// TIA Portal V20 export
// export: Created 2025-12-01T14:57:26.5426352Z, ExportSetting None, DisplayName Totally Integrated Automation Portal, DisplayVersion V20 Update 3, DisplayName TIA Portal Openness, DisplayVersion V20 Update 3, DisplayName TIA Portal Version Control Interface, DisplayVersion V20 Update 3, DisplayName STEP 7 Professional, DisplayVersion V20 Update 3, DisplayName STEP 7 Safety, DisplayVersion V20 Update 2, DisplayName WinCC Basic/Comfort/Advanced, DisplayVersion V20 Update 3, DisplayName WinCC Professional, DisplayVersion V20 Update 3, DisplayName WinCC Unified, DisplayVersion V20 Update 3
FUNCTION "FC600_ini+ref_dato_encoder_NEW" : Void   // FC600, LAD
{ S7_Optimized_Access := 'FALSE' }
// stored: AutoNumber false, SetENOAutomatically false
   VAR_INPUT
      Detector_referencia : Bool;
      ID_Quimarox : UInt;
      dato_encoder_actual : DInt;
      V_cnt_tout_refresco : UDInt;
   END_VAR
   VAR_IN_OUT
      m_aux_pf_detect : Bool;
      MEM_CNT_TOUT : UDInt;
   END_VAR
   VAR_TEMP
      fp_detector : Bool;
      tout : Bool;
      fecha : Date_And_Time;
      retval : Int;
      hora : Time_Of_Day;
   END_VAR
   VAR_TEMP   // added for the SCL form of the ladder/FBD networks
      _w1 : Bool;
   END_VAR
BEGIN

REGION Network 1
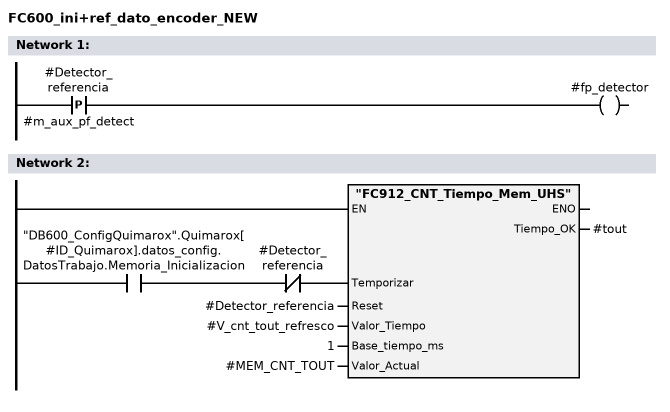
   RUNG wire#powerrail
      P_Contact(operand := #Detector_referencia, bit := #m_aux_pf_detect)
      Coil( #fp_detector )
   END_RUNG
   // the same network as SCL:
   #_w1 := #Detector_referencia AND NOT #m_aux_pf_detect;   // rising edge of #Detector_referencia
   #m_aux_pf_detect := #Detector_referencia;
   #fp_detector := #_w1;
END_REGION

REGION Network 2
   RUNG wire#powerrail
      "FC912_CNT_Tiempo_Mem_UHS"(Temporizar := wire#w1, Reset := #Detector_referencia, Valor_Tiempo := #V_cnt_tout_refresco, Base_tiempo_ms := 1, Valor_Actual := #MEM_CNT_TOUT, Tiempo_OK => #tout)
   END_RUNG
   RUNG wire#powerrail
      Contact( "DB600_ConfigQuimarox".Quimarox[#ID_Quimarox].datos_config.DatosTrabajo.Memoria_Inicializacion )
      I_Contact( #Detector_referencia )
   END_RUNG wire#w1
   // the same network as SCL:
   "FC912_CNT_Tiempo_Mem_UHS"(Temporizar := "DB600_ConfigQuimarox".Quimarox[#ID_Quimarox].datos_config.DatosTrabajo.Memoria_Inicializacion AND NOT #Detector_referencia,
                           Reset := #Detector_referencia,
                           Valor_Tiempo := #V_cnt_tout_refresco,
                           Base_tiempo_ms := 1,
                           Valor_Actual := #MEM_CNT_TOUT,
                           Tiempo_OK => #tout);
END_REGION

NETWORK
TITLE = 

      SET;
      A     "DB600_ConfigQuimarox".Quimarox[#ID_Quimarox].datos_config.DatosTrabajo.Memoria_Inicializacion;
      JC    NXT;

      SET;
      AN    #fp_detector;
      JC    fin;


NETWORK
TITLE = 
//====================================================================================================================================================================================
// primera actualización del dato del encoder. Ademas de memorizar cual es el dato del encoder en este momento y pasarlo a la memoria, registramos la hora en al que se ha producido

      L     #dato_encoder_actual;  //en el primer ciclo giramos en vacio hasta que detectemos el elemento para referenciar
      T     "DB600_ConfigQuimarox".Quimarox[#ID_Quimarox].datos_config.DatosTrabajo.Memoria_Dato_Encoder;

      SET;
      =     "DB600_ConfigQuimarox".Quimarox[#ID_Quimarox].datos_config.DatosTrabajo.Memoria_Inicializacion;

      CALL  RD_SYS_T
      ( RET_VAL := #retval,
        OUT     := #fecha
      );

      CALL  T_CONV
      ( IN  := #fecha,
        OUT := #hora
      );


      L     #hora;
      T     "DB600_ConfigQuimarox".Quimarox[#ID_Quimarox].datos_config.DatosTrabajo.Hora_Ultimo_Refresco;  //#Hora_ultimo_refresco

      BE;

//===============================================================================================================================================================================

NETWORK
TITLE = 
NXT:  A     #fp_detector;
      JC    REF;

      BE;


NETWORK
TITLE = 
//==================================================================================================================================00
REF:  L     #dato_encoder_actual;
      T     "DB600_ConfigQuimarox".Quimarox[#ID_Quimarox].datos_config.DatosTrabajo.Memoria_Dato_Encoder;

      CALL  RD_SYS_T
      ( RET_VAL := #retval,
        OUT     := #fecha
      );

      CALL  T_CONV
      ( IN  := #fecha,
        OUT := #hora
      );

      L     "DB600_ConfigQuimarox".Quimarox[#ID_Quimarox].datos_config.DatosTrabajo.Hora_Ultimo_Refresco;  //#Hora_ultimo_refresco
      T     "DB600_ConfigQuimarox".Quimarox[#ID_Quimarox].datos_config.DatosTrabajo.Hora_Anterior_Refresco;
      L     #hora;
      T     "DB600_ConfigQuimarox".Quimarox[#ID_Quimarox].datos_config.DatosTrabajo.Hora_Ultimo_Refresco;  //#Hora_ultimo_refresco


      BE;

fin:  BE;
END_FUNCTION
